// TIA Portal V20 export
FUNCTION_BLOCK "Dancer"   // FB19, LAD
// stored: MemoryReserve 100, Namespace Unit1.Em3, SetENOAutomatically false
   VAR
      instLConSMC_RFG { S7_SetPoint := 'True'} : "LConSMC_RFG";
   END_VAR
BEGIN

REGION Network 1
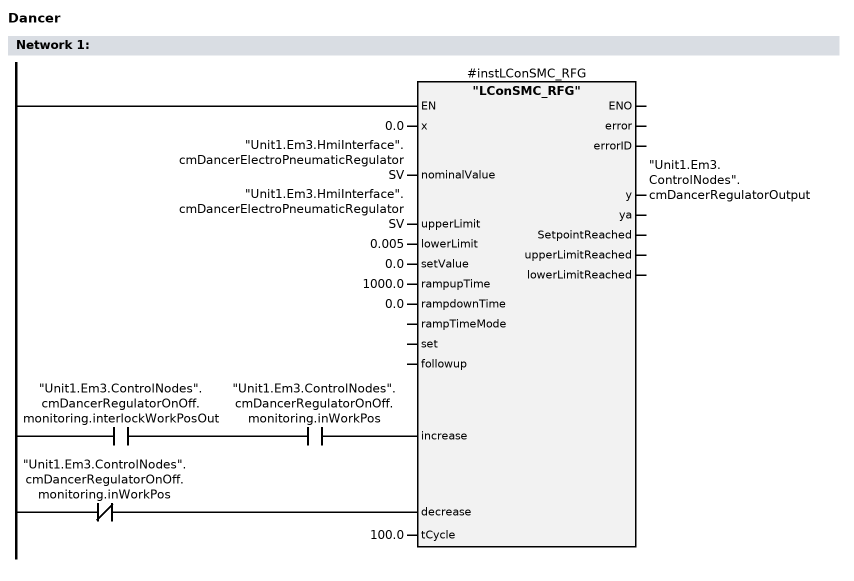
   RUNG wire#powerrail
      #instLConSMC_RFG(increase := wire#w1, decrease := wire#w2, x := 0.0, nominalValue := "Unit1.Em3.HmiInterface".cmDancerElectroPneumaticRegulatorSV, upperLimit := "Unit1.Em3.HmiInterface".cmDancerElectroPneumaticRegulatorSV, lowerLimit := 0.005, setValue := 0.0, rampupTime := 1000.0, rampdownTime := 0.0, rampTimeMode :=, set :=, followup :=, tCycle := 100.0, error =>, errorID =>, y => "Unit1.Em3.ControlNodes".cmDancerRegulatorOutput, ya =>, SetpointReached =>, upperLimitReached =>, lowerLimitReached =>)
   END_RUNG
   RUNG wire#powerrail
      Contact( "Unit1.Em3.ControlNodes".cmDancerRegulatorOnOff.monitoring.interlockWorkPosOut )
      Contact( "Unit1.Em3.ControlNodes".cmDancerRegulatorOnOff.monitoring.inWorkPos )
   END_RUNG wire#w1
   RUNG wire#powerrail
      I_Contact( "Unit1.Em3.ControlNodes".cmDancerRegulatorOnOff.monitoring.inWorkPos )
   END_RUNG wire#w2
   // the same network as SCL:
   #instLConSMC_RFG(x := 0.0,   // "LConSMC_RFG"
                    nominalValue := "Unit1.Em3.HmiInterface".cmDancerElectroPneumaticRegulatorSV,
                    upperLimit := "Unit1.Em3.HmiInterface".cmDancerElectroPneumaticRegulatorSV,
                    lowerLimit := 0.005,
                    setValue := 0.0,
                    rampupTime := 1000.0,
                    rampdownTime := 0.0,
                    increase := "Unit1.Em3.ControlNodes".cmDancerRegulatorOnOff.monitoring.interlockWorkPosOut AND "Unit1.Em3.ControlNodes".cmDancerRegulatorOnOff.monitoring.inWorkPos,
                    decrease := NOT "Unit1.Em3.ControlNodes".cmDancerRegulatorOnOff.monitoring.inWorkPos,
                    tCycle := 100.0,
                    y => "Unit1.Em3.ControlNodes".cmDancerRegulatorOutput);
END_REGION
END_FUNCTION_BLOCK
